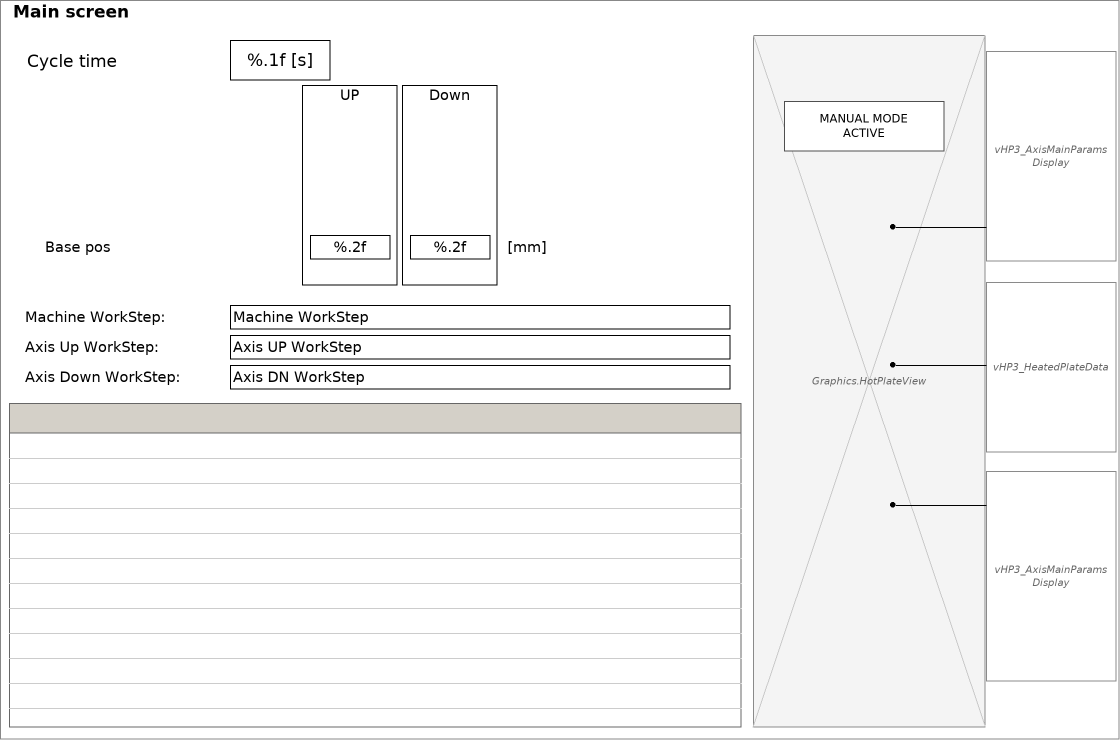
VISUALIZATION vHP3_MachineSub_Main_Old  // 1120x740
VAR_IN_OUT
	fbHP: fbHPv3_Control;
END_VAR
    Image (753,35 232x692), image: Graphics.HotPlateView
    Frame (986,51 130x210)
        shows vHP3_AxisMainParamsDisplay(fbAxis := fbHP.fbAxisUp)
    Frame (986,471 130x210)
        shows vHP3_AxisMainParamsDisplay(fbAxis := fbHP.fbAxisDn)
    Frame (986,282 130x170)
        shows vHP3_HeatedPlateData(fbHP := fbHP)
    Ellipse (890,224 5x5)
    Line (896,227) (986,227)
    Ellipse (890,362 5x5)
    Line (896,365) (986,365)
    Ellipse (890,502 5x5)
    Line (896,505) (986,505)
    Rectangle (784,101 160x50), "MANUAL MODE ACTIVE", invisible if: NOT fbHP.bManualMode
    RoundedRectangle (10,0 300x26), "Main screen"
    Table (9,403 732x324), data array: fbHP.fbTimeStats.astTT
        p3854506369: fbHP.fbTimeStats.astTT[INDEX].sStepName
        p1892666644: fbHP.fbTimeStats.astTT[INDEX].rStepTime
        p2232123230: Step name
        p511219082: Step time
        p1128707560: fbHP.fbTimeStats.uiTTLastIndex
    Label (42,235 260x24), "Base pos"
    RoundedRectangle (402,85 95x200), "Down"
    RoundedRectangle (302,85 95x200), "UP"
    Rectangle (310,235 80x24), "%.2f", text variable: fbHP.fbAxisUp.lrBasePos_mm
    Label (502,235 50x24), "[mm]"
    Rectangle (410,235 80x24), "%.2f", text variable: fbHP.fbAxisDn.lrBasePos_mm
    Label (22,305 200x24), "Machine WorkStep:"
    Label (22,335 200x24), "Axis Up WorkStep:"
    Label (22,365 200x24), "Axis Down WorkStep:"
    Rectangle (230,305 500x24), "Machine WorkStep", text list: 'tlHPv3', text index: 0
    Rectangle (230,335 500x24), "Axis UP WorkStep", text list: 'tlHPv3', text index: fbHP.fbAxisUp.iHMI_StepName
    Rectangle (230,365 500x24), "Axis DN WorkStep", text list: 'tlHPv3', text index: fbHP.fbAxisDn.iHMI_StepName
    Rectangle (230,40 100x40), "%.1f [s]", text variable: fbHP.rCycleTime_s
    Label (24,41 204x40), "Cycle time"
END_VISUALIZATION

(* stored: Version 1.1.0.1, ProductVersion 3.1.4024.12
   Visu vHP3_MachineSub_Main_Old: Id {c4f4155f-f6ad-4462-a550-b682a13439b7} *)
